FUNCTION_BLOCK F_FIND (* find the character position of the beginning of the first occurrence of IN2 in IN1, no occurrence returns 0 *)
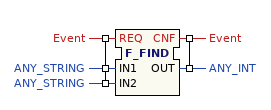
  EVENT_INPUT
    REQ WITH IN1, IN2; (* Service Request *)
  END_EVENT
  EVENT_OUTPUT
    CNF WITH OUT; (* Confirmation of Requested Service *)
  END_EVENT
  VAR_INPUT
    IN1 : ANY_STRING; (* input string 1 *)
    IN2 : ANY_STRING; (* input string 2 *)
  END_VAR
  VAR_OUTPUT
    OUT : ANY_INT; (* number of occurrence *)
  END_VAR
END_FUNCTION_BLOCK
